# EPICS autosave request: ADPvCam/iocs/pvcamIOC/iocBoot/iocPvCam/auto_settings.req
file "pvCam_settings.req",  	    P=$(P),  R=pvcam:
file "NDStdArrays_settings.req",  P=$(P),  R=image:
file "commonPlugin_settings.req", P=$(P)
